(* IEC 61131-3 sources: advent-of-code/day10, 6 files *)

(* ---- demo.st ---- *)
VAR_GLOBAL CONSTANT
	str_len : DINT := 24; //Max length
	input_size : DINT := 9;
END_VAR

VAR_GLOBAL
	input : ARRAY[0..input_size-1] OF STRING[str_len];
END_VAR

FUNCTION set_input : __VOID
VAR_TEMP
	c : DINT;
END_VAR
	input[c] := '[({(<(())[]>[[{[]{<()<>>'; c := c + 1;
	input[c] := '[(()[<>])]({[<{<<[]>>('; c := c + 1;
	input[c] := '{([(<{}[<>[]}>{[]{[(<()>'; c := c + 1;
	input[c] := '(((({<>}<{<{<>}{[]{[]{}'; c := c + 1;
	input[c] := '[[<[([]))<([[{}[[()]]]'; c := c + 1;
	input[c] := '[{[{({}]{}}([{[{{{}}([]'; c := c + 1;
	input[c] := '{<[[]]>}<{[{[{[]{()[[[]'; c := c + 1;
	input[c] := '[<(<(<(<{}))><([]([]()'; c := c + 1;
	input[c] := '<{([([[(<>()){}]>(<<{{'; c := c + 1;
	input[c] := '<{([{{}}[<[[[<>{}]]]>[]]'; c := c + 1;
END_FUNCTION

(* ---- input.st ---- *)
VAR_GLOBAL CONSTANT
	str_len : DINT := 150; //Max length
	input_size : DINT := 110;
END_VAR

VAR_GLOBAL
	input : ARRAY[0..input_size-1] OF STRING[str_len];
END_VAR

FUNCTION set_input : __VOID
VAR_TEMP
	c : DINT;
END_VAR
input[c] := '<([<({{[<{{((<()>({}{})}<({}<>)>)}}>[<{(([()<>]<<>{}>))}<{({<>[]}<<>>)[([]<>)<{}{}>]}>>]]}}[<[{{[{{[<><>]'; c:= c+1;
input[c] := '[<{{{[((({<<<[()[]]{()()}><{<><>}(<>{})>><<{<><>}{{}[]}>{(()())[[]{}]}>>{[[(<>[]){<>{}}][(()())(()[])]]'; c:= c+1;
input[c] := '(((<{<[[<[{(((<><>)[{}{}]){{{}<>}[()<>]})(([<>()][<>{}]){{[]()}})}[({([][])<{}<>>}{[[]<>]{()'; c:= c+1;
input[c] := '[(<{<[<<<<[[{<[]()><<>()>}[{{}<>}<()>]]<<[[]{}]>{({}())}>]((((<>())<(){}>)<{[]{}}<(){}>>)[{[[]<>]<['; c:= c+1;
input[c] := '[[{(<{<<[{(<({<>{}}<()[]>){<<>[]>{<>}}><[[()[]]]{{()<>}{()<>}}])[{[(<>())]<<[]{}>(<>[])>}<[{'; c:= c+1;
input[c] := '(<<<[[<{({<<([{}{}](<><>)){{<><>}(())}>{<{(){}}{[][]}>[{[][]}([]())]}><([{{}[]}[[]{}]](<[]{}><{}<>>))((<(){'; c:= c+1;
input[c] := '<<<{((<<{[([<[[]{}]([][])>{[<>()][[][]]}]<<[()[]][[]{}]>[<<><>>(<><>)]>)<({{{}<>}{{}}}{{<><'; c:= c+1;
input[c] := '{[(<[{{{<[{({([]{}){{}{}}}[({}<>)])[([()[]]<[]{}>)<[{}{}]{{}()}>]}(<{{{}<>}(()[])}>{{<()<>><[]<>>}'; c:= c+1;
input[c] := '[<<{({[{((({<<<><>>(()())>{{[][]}<{}()>}}[[((){})[{}()]]<[()<>]>]){{(<{}<>>[()<>]){{[][]}(()<>'; c:= c+1;
input[c] := '({[([([<(<<[{<<><>>({}())}[[(){}][[][]]]]>><<(({<><>}{[][]})<{()()}[[]<>]>)[{((){}){{}[]}}(<<>()>{{}()})]><<'; c:= c+1;
input[c] := '[[[{[<({{<[[[<{}{}>(()())]{(<>[])([][])}]({{(){}}})]<[<{{}[]}{()}>[{<><>}]][<((){})([][])>]'; c:= c+1;
input[c] := '[(<{<{(<<<<{{[[][]]<()[]>}){{<<>{}>}}>({[(()())(<>[])]}(<{()()}[<>]>{[[]]<<>()>}))>(<[{({}{})}][{[{}()]'; c:= c+1;
input[c] := '<(<<[([[((<<{<[]{}>{{}<>}}(({}())[[]{}])>(<{<>()}[()()]>>>))]{<{{<(<()<>>{{}()})([{}<>](<><>))>'; c:= c+1;
input[c] := '[{[<[([[<[((([()[]]<{}{}>))<{[{}()][(){}]}([{}<>]<()<>>)>)]>[{((([{}()]{()()>)<(<><>)(()[])>)[(([]()'; c:= c+1;
input[c] := '{[{[{<<([({<<[{}()]<()<>>>{[[][]]({}())}>}[[<{{}<>}{<>}>]])(<<{[()[]]}(((){})({}{}))>[({{}()})]>)]('; c:= c+1;
input[c] := '({{{<<<<(([([[<><>]<<>[]>]{<()<>><()[]>})<([<>{}])>])(<<{{()}<()[]>}<([]<>)>>{{[{}()][[]<>]}[{<>}{()()'; c:= c+1;
input[c] := '[{(([{<{{(<{<<[]()>{{}<>}>}[<({}[])<{}<>>><{<>()}>]>)}<{{{{<<>{}>{()()}}}[[{()()}(()<>)><<{}<>>>]}[[(<(){}>('; c:= c+1;
input[c] := '[[{<[<(<[[<<({{}()}{{}})(({}{})[[]{}])>[([<>{}]({}<>))])]{<[<[[][]]<()<>>>]{([()()]{<><>})<{[]{}}[[]()]>}><'; c:= c+1;
input[c] := '([<<{({[({[({<{}[]>{{}<>}}){<[<>[]]>[(()())]}]{{{{{}[]>{()<>}}}<[{{}<>}<[]()>]([<>]<<><>>)>}})'; c:= c+1;
input[c] := '(([<[[{{(<[{{(()<>)}<<{}()>{<>{}}>}<[<[]()>[()()]]([<>()]{()})>)[(<[<><>]{{}<>}>{{{}()}{[]()}})<'; c:= c+1;
input[c] := '[([[[([[[<[{{<()()>{[][]}}(<[][]>)}[{<{}()>{<>[]}}]]>({[[{<><>}<[][]>]([()]{()[]})]}{([<<><>>[{}('; c:= c+1;
input[c] := '(<({<[[[[(((({[]{}}<{}<>>)[<(){}>[()<>]])){<(<<>{}>)<<()<>><()[]>>>{[[()()]<[][]>][{{}()}<<>{'; c:= c+1;
input[c] := '{{{{[[<{<{(<(([]())[{}[]])<(()<>){{}{}}}>){{{<{}[]><{}<>>}{(()[])[<><>]}}<{{()()}<<>[]>}>}}><(<[(<{'; c:= c+1;
input[c] := '<<[(<<<([{<{(({}())[{}[]])(<(){}>(<><>))}>([[(<>[])(<>[])]<({}{})<{}>>](((<>())<{}[]>)[[<>'; c:= c+1;
input[c] := '<{{((([[<{[(({<>{}}({}())))[([[]()][{}{}])]]}(([<([][])<<>()>>]<{{<>[]}(()())}[({}())[()()]]>)'; c:= c+1;
input[c] := '(({[{[[[[(<<[[(){}][(){}]]<{()<>}<[][])>>{({[][]}{<>{}}){<[][]>}}><{(([]{}){{}<>}){[()<>][('; c:= c+1;
input[c] := '{<[[<<([<{<<{[<>{}}{<><>}}(({}()))>[[{[]()}](<<>>{<><>})]><<([<>{}]{[][]})[<{}[]>{<><>}]>>}{[{(<<>()><{}<>'; c:= c+1;
input[c] := '({{{((({<<({<[<>()](()[])]}){((<{}()>{[]<>}){<[]{}>[[][]]})<[[[]{}](())](<{}<>>[{}])>}>[{{[(<>[])]}[<({}{'; c:= c+1;
input[c] := '{<(<[{({[[[{[[{}<>][(){}]]{{(){}}}}<<[[]()]{<>}><[{}[]]>>]{<<((){})[{}]>({<><>}{()[]})><<[{}()]{'; c:= c+1;
input[c] := '[[[(({<((<({<<{}>>}<[([]{})[[]]]>)<<{[()[]](<><>)}><<{[]{}}[[]]>{{()[]}{[]()}}>>><[((<(){}'; c:= c+1;
input[c] := '{{<{{{<<{<{<((<>[])<()[]>)<(<>{}){[][]}>><(({}<>){[][]}){[()<>]{<>{}}}>}>[((<<(){})({}())><([]'; c:= c+1;
input[c] := '[[[{({<[{[[<<(()<>)({}())>({<><>}[<><>])>]]<(<{<()<>>([]())}{[[]<>]{<>()}}>{<([][])((){})>([{}][()<>])})>}]<('; c:= c+1;
input[c] := '<<{[{[[<([[<<[{}<>]>[({}())<()[]>]>[{<(){}><{}<>>}[<<>>({}{})]]]<<{<()[]><()()>}({{}()}[{}<>])>>]<<([([]('; c:= c+1;
input[c] := '{<<<(<{{[{{{<<{}[]>{()()}>{[<>[]]({}())}}}<[<([]())>{<()()>(()())}][<(()())<{}<>>>((<><>)[[][]]]]>'; c:= c+1;
input[c] := '[[[({<(([[(<({()<>}<[]<>>)>[({[]}{<><>})<<(){}>{<><>}>])]]<(<[<<()()]<{}()>>(<{}()>([][]))]<<{<><>}>>>){'; c:= c+1;
input[c] := '<<[[<({<({[<{(()[])}{{[]()}<[]{}>}>]<[(<[]{}><<>{}>)<[()[]]([]{})>]>})>((<([<[<><>]([]{}}><{<>()}<()[]>>]{'; c:= c+1;
input[c] := '({[[[{{([[((<<{}<>}[{}<>]>)(({{}<>}<()()>)[[[]<>]<()<>>]))<(<{[][]}>)<{{[]<>}<[]<>>}[(<><>){(){}}]>>][<'; c:= c+1;
input[c] := '{<[[[[[<[[{{{{()}[[][]]}[<(){}>[[][]]]}(<[{}{}]>)}(<<<()()>{<>}>>)]<([[[()<>]((){})]([[]()]<{}{}>)]([{{}('; c:= c+1;
input[c] := '[<(({(((<[(<<[[]{}][<><>]>[{(){}}[[]]]><{{()[]}<<>()>}{{()}{(){}}}>)(<[([]())]<{{}{}}(())>>)]([([{()[]}[['; c:= c+1;
input[c] := '(({[([{{((({{<<>[]>}}<([{}[]][[]()])[{{}[]}<<>{}>]>)<({([])<[]{}>}){(((){})[<>[]]){<<>[]>[{}()'; c:= c+1;
input[c] := '<{<{(<<({([([([]())(<>[])][{()<>}{<>{}}])](({<()()>{()<>}}{{[]}[[][]]})[[[{}{}][()[]]]])]}(({[[{<>()}[{}()]'; c:= c+1;
input[c] := '[[{[{{[({<{<(<{}<>>)[[{}{}>[<><>]]>[((())([]<>)){([]())<<><>>}]}>{{{<{<>[]}({}{})>{([]{}){[][]}}}[{{<>'; c:= c+1;
input[c] := '[[{[<([{([<<<(<><>){[]{}}>{{[][]}([]<>)}>><{<<<>()>{<><>}>[<[][]>([]())]}({[{}[]]{<>()}}({()()}(()<>)))>])}])'; c:= c+1;
input[c] := '{{<((([<[({{(([]){[][]})[(()<>)<()()>]}{{{()[]}}([()[]][{}{}])}})<{({[()[]]<[]{}>}[<()()><()[]>])'; c:= c+1;
input[c] := '([<<<([{{<({{[{}<>][<>()]}{([]<>){(){}}}}){({<{}()>}[(()){<><>}])}><{<(<()[]>({}{}))(({}{})'; c:= c+1;
input[c] := '{{[([<[{<<{<{[{}[]][(){}]}[[[]()]{()[]}]>}><[(([<>{}]){{<>()}{()<>}}){[{<>{}}[[]<>]]{<[]<>>}}][[[{[]<'; c:= c+1;
input[c] := '{<<<<{(((<{([{{}{}}][[[]()]<<>()>])<([()<>]([]))[[<><>][{}()]]>}{<{{(){}}<()<>>}<{<>{}}{<>()}>>(<{'; c:= c+1;
input[c] := '<[({<{{{<((<<({})([]<>)>((<>[]){[]()}}>)(<[<(){}>({}[])]>[<({}<>){[][]}>[{()<>}<<><>>]]))>[({[([<>{}][{}()])<'; c:= c+1;
input[c] := '(({[[{<{[[((<[<>()]><{()<>}[[]<>]>)([{[]()}[[]()]](({}{}){<>()})>){<{(()())(<>[])}[<()[]>[()()]'; c:= c+1;
input[c] := '[(([{{<{<[{{{[{}{}]<(){}>}[<[]{}>({}())]}({[()[]]{[]()}}[<{}[]>(<>)])}[{{<[]{}>(()<>)}<[[]()]<<>[]>)}<<<<>()'; c:= c+1;
input[c] := '<(<<{<([([(<[{{}<>}<()()>][{()[]}(<><>)]>{{<[]<>><{}[]>>{{{}}{[]<>}}})({[<[]{}>[[][]]]}{{<'; c:= c+1;
input[c] := '((<<<([[<<{([<<>{}>{<>()}])<<{[]{}}[()[]]>>}[<{([]())[<>{}]}>{((()[]){{}<>))[<()<>>([]<>)]}]>{(({[[]]'; c:= c+1;
input[c] := '{<<((({({[<[[[<><>][<>{}]]{({}<>)<()[]>}][<<[]{}}<[]()>>[[[]<>]]]>([[[{}{}]]<<<><>><<>{}>>'; c:= c+1;
input[c] := '[{<([{{<{(<{{{(){}}{{}[]}}(<<>()>[()[]])}{{{{}}(()())}{[()<>]}}>[{[{[][]}{{}<>)]}((((){}){[]{}})(({})<<>{}'; c:= c+1;
input[c] := '[{[(<[{<{{[<{{()()}{()[]}}<<()()><{}[]>>>][<({()()}[()[]]){([][])[<>{}]}>(((()()))((<>{})<{}{'; c:= c+1;
input[c] := '(<(<([<<<{[<({<>}{()()})><((<>))<<{}[]><<><>>>>]{<{[[][]]}{{[]{}}{[]<>}>>[[[[]()]({})]]}}><<<<'; c:= c+1;
input[c] := '<([<(<<<(({{<[<><>]<[]<>>>(<[]()>[{}<>])}[<(()()){{}<>}>]}))<<[{{[<>[]]<()[]>}{(()<>){()()'; c:= c+1;
input[c] := '<[(<{{[[[<(([[<>()]([][])])){{{[()()]{{}[]}}[([]{}){(){}}]}{[<[]>{[]()}][[<>]({}())]}}>]]<(<[{<{<>()}{()['; c:= c+1;
input[c] := '<{{{[(<{<[<{{<()>(<>{})}[({}()){()()}]]([{<>{}}[()()]](<[]<>><<>{}>))>[<{<[]()>(<>)}<{[]{}}[('; c:= c+1;
input[c] := '<{(<[<[<{<({<[<><>}[[]()]>}([<(){}><<><>>][<()()><<><>>]))([[([]())<{}>]<[()()]{<>{}}>]{(({}'; c:= c+1;
input[c] := '<(<({(<[<[(((<<>{}>{{}()})){{[[]()](())}{{<><>}<<><>>}})([<<()()><[]())>[[<>()]<<>[]>]][<{()()}'; c:= c+1;
input[c] := '((<[{{(<[([<([()()](<>{}))(<{}()>[{}{}])>({<{}{}>(<>[])})])]>)}<({((([(<[]{}>({}[]))]{((<><>)(()()))}))(({{<{'; c:= c+1;
input[c] := '{({[<<[(<<((<<{}[]>[()<>]>{<<>[]>{[]()}}){[<<><>>[()[]]]<<{}()>[()<>]>})[{[{{}<>}{()}]}<(<()[]><{}{}>)[['; c:= c+1;
input[c] := '{{[<((<((<{[([[][]]<{}<>>)((()[]))]}>{[{(({}())[()[]]){{[][]}([][])}}](<<[<><>]{<>}><<{}<>><[][]>>>'; c:= c+1;
input[c] := '[[[<(<{{([{(<(<>{})(()<>)><(<>[])[{}()]>)([[[]()][[]<>]])}[[{<[]()>(<><>)}[(()){<>()}]]({{[]()}})]])[['; c:= c+1;
input[c] := '<({([{(<{{[<<[(){}][[]()>>[[{}{}](()[])]>]{{[[{}<>]{{}<>}]{({}<>)[{}{}]}}[({()()}[{}<>]){((){})}]}}{{[[{{'; c:= c+1;
input[c] := '[[[[{<[<(([<[<[]{}><<>{}>]<<[]<>>(()[])>>([(<>)<{}()>])])<{{({[]{}}{[]()})}<[[<><>]{[]<>}]{<<>()><<>()>}>'; c:= c+1;
input[c] := '<<<[([[(({(<[<{}>[{}()]]{{()}(()[]}}>(<<<>()>(<>[])>))<<[{<>()}{<>[]}][{[]{}}<{}[]>]>>}){<<<(<<>'; c:= c+1;
input[c] := '{{<[{{({{(([[([]{})<{}()>]]))){(<{{<<>[]>(<>[])}<<()><[]<>>>}>([([<>()]<{}[]>)(({}{}))]<<([]())[<>'; c:= c+1;
input[c] := '([<[({[{{[[[({<>{}}<(){}>)({<>[]}{()<>})](([(){}]{[]()}))]<[<(<>[])({}<>)>][[[[]{}]<()>]<<<>[]>{[]<>}>]>]'; c:= c+1;
input[c] := '{[{[[{<(<<({{([]<>)([]{})}<<{}<>><<>[]>>}(({()()}[{}()]){(<><>)[<>[]]]))<<[([])(<>[])]{([]())('; c:= c+1;
input[c] := '({<<{{[<<[{{<[(){}][[]]><{[]()}<[]{}>>}[<<<>()>{{}()}>[<{}<>>[<><>]]]}](<<[(<>{})[()]}{<<>><[]'; c:= c+1;
input[c] := '<<<([{[([{{[{[[]<>][<>[]]}]}{<([[][]]){[<>[]]<{}()>}><(<[]<>>(<>{}))[<[][]>{<>}]>}}{<{{[<>{}]{()'; c:= c+1;
input[c] := '<((<([([<{<[([{}<>](<>()))<([]<>)([]<>)>][<{()<>}{[]<>}>]>}<{[(<[]()>(<><>))[<(){}>[[][]]]](<([]())<<>[]>>['; c:= c+1;
input[c] := '{[<[<<{{(<{[{((){})<{}[]>}[([][])]]}{[({()<>}){[{}<>](<>{}))]}>)}<[[(<(<()<>>){(()())([]{})}>({[{}[]]'; c:= c+1;
input[c] := '<([[<({{[<({[({}{}){{}()}]<((){})[<><>]>})([[{[][]}<()<>>]<[()<>][{}{}]>])>]}}){{[(({(({[]()}{()()}'; c:= c+1;
input[c] := '<({([<[{(<[{(({}[]))}[[{[]<>}{{}[]}](({}[]))]]<[[(()[])[()()]]{[{}()>}]>>{<<{[[]<>](()())}[<{}[]>(<>'; c:= c+1;
input[c] := '(([[<(<<[{<(<[{}{}]{()<>}>)((<(){}>([]))({<>{}}[<>[]]))>(<<{()[]}{(){}}>[[<>()]]>[<{()[]}<()[]>>{({}<>){[]<'; c:= c+1;
input[c] := '{<[<<{(<{{<[{[{}()][<><>]}][{({}{})(<>[]))]>{<[[<><>]]<<<>()>({}[])>>({<[]<>>([]<>)}{[(){}]([]{})})'; c:= c+1;
input[c] := '{{<((([<{(([{[<>{}]{{}<>}}])<<<{<>[]}{(){}}>{(()[])[()[]]}>{{<<>()>}([(){}]{{}<>})}>)}{(([{{{}[]}(<>())'; c:= c+1;
input[c] := '{[(<{{{<[[{{[[()[]](<>{})]((()<>)({}[]))}}]][{([[{{}[]}<[]<>>]][{(<>{})}[(<>()){<><>}]])}>>[(['; c:= c+1;
input[c] := '<<<{([((<<{(({{}{}}({}{})))}{(<(<><>)[[]<>]>{[{}[]](<>)})<{{<>()}{{}<>}}<<<>[]><<>()>>>}>>))]){'; c:= c+1;
input[c] := '<{(<[[(({<[{{<<><>><{}<>>}<<<>{}>{()()}>}]>}))[((([([{[]{}}]([{}()][<><>]))(((<>())(<>]))]['; c:= c+1;
input[c] := '([<<[({(({{((<[]{}>{()[]}})({[<><>][<>()]}(<<><>>[[]()]))}{{{(()<>)({}{})}(<{}()><[]()>)}{{{<><>}'; c:= c+1;
input[c] := '[<<<{{<<{<{<<[()()](<><>)>>([({}){{}[]}]{<[]()>{{}()}})}<[{([]())<{}<>>}([{}()]<{}[]>)]<(<[]'; c:= c+1;
input[c] := '{{<[({({<{({((()<>)){[[]()]<(){}>>}<[[{}]{<><>}]<(()<>)<()()>>>)}(({((<><>)[{}[]]){[[]()][()[]]}})<({'; c:= c+1;
input[c] := '<[{<({<({(({{<(){}>[[]{}]}<<[][]><{}{}>>})[(([{}()][<>()]))[(<<>{}>([][]}){[[]{}]}]])[<[{(()<>)[{}<>]}]>]'; c:= c+1;
input[c] := '([(([{<(<{[<{([][]){[][]}}(<<>><[]{}>)>({[<>()]{{}<>}}(<<>[]>{<>{}}))][({{[]()}{[]}}(([]{})(()<>))'; c:= c+1;
input[c] := '<{<<<({[[(<<{(()<>)[[]{}]}<<()()>>>><[({()[]}[[][]]){<[][]>(<><>)}][(({}{})<()[]>){{{}()}<[]{}>}]>)[<((([]{}'; c:= c+1;
input[c] := '<([[([<<<{<<<<<><>>({}())>{{[]()}[{}[]]>>[<[<>()]({}{})>]>(({<{}{}>{<>{}}}{<{}[]>{{}()}}){[<[]()>{()<>}'; c:= c+1;
input[c] := '[{{<{[{{{<{{<([][])[()<>]>{{[]{}}({}())}}((<<>[]>([][])))}><{<<<{}<>><<>()>>{(()<>){[]{}}}>}{([{[][]}{<>{}}])'; c:= c+1;
input[c] := '[({<((({(<{[{<[][]}(<>[])}<<{}<>>{{}<>}>]({{<>()}[{}{}]})}(<{{{}()}<<>[]>}[([]{})<[][]>]>[{(<>'; c:= c+1;
input[c] := '<([[[<{{<<<[(((){})(()()))([<><>]{()})]<<[<>]([])>(([]<>))>>{{[<()>]<(()[])([][])>}[({{}}<{}{'; c:= c+1;
input[c] := '{<<((<[{<{<[{[[][]]{<><>}}{<(){}>{<><>}}]<((<>{})<<>[]>)>>((((<>[]){[]()})({<>()}))([[{}[]]{<>[]}]<'; c:= c+1;
input[c] := '(<{(<[[([[([<({}{})[()<>]>])][<{<({}())><{()()}>}>{[{[{}<>]([])}](([()()]))}]])]]>)}>[[({{'; c:= c+1;
input[c] := '(<[[[{<{[<([{({}{}){{}()}}[(<>{})<()()>]][{{{}()}}<{<>[]}[()<>]>]){{((<><>){()<>])<<<>()>[{}['; c:= c+1;
input[c] := '<{<<[((<<<{([{{}<>}({})]{((){})[[]<>]})<[[()<>]([]())](<[]<>>({}<>))>}{(<{()[]}>{<[]<>>})<'; c:= c+1;
input[c] := '{[([<[<[({{[<[<>()][{}[]}>((<>())<[]<>>)]{(<{}<>>(()()))([()()])}}}<(<(<<>{}>{<>{}})><({[]{}}['; c:= c+1;
input[c] := '{{[[[<<<<[[{({[]<>}<()()>)<<(){}>{<><>}>}{[([]<>)[<>[]]]}]{<[{()()}(<><>)]{{<>{}}<[]{}>}>((<{}()>{(){}}))}>>>'; c:= c+1;
input[c] := '({[<[[<{<([<<<()<>}<{}{}>>(<<>[]>(<>()))><{[<>()]({}<>)}<{[]{}}>>])>}{{{<{({[]{}}<<>>)<<[]<>'; c:= c+1;
input[c] := '([((((<(<[({((<>())<()<>>)}([<{}()>{<>()}]{{{}()}{[]<>)}))([<(<>{})><[(){}][<>()]>](([()]<[]{}>)(<{}{}>{()'; c:= c+1;
input[c] := '{[(<{({(<([(<[{}()][{}()]>)[[[{}()](()())]<{[][]}<[]<>>>]][({[()()]{{}{}}}((<><>)(<>())))<<{()()}{[]{}}}[{[]'; c:= c+1;
input[c] := '<([[{<<{<<{(([()<>]{<>[]})<<[][]>({}[])>)({<{}{}>([]<>)})}{<{{[][]}{[]{}}}[((){})((){})]><([[][]]){{()()}}>}'; c:= c+1;
input[c] := '(([<[[[(({{[[[[][]](<>())]{<<>><<>()>}]<<(()<>)>[<<>{}>{<><>}]>}[<(<<><>><{}{}>)[<()<>><[]()>]>[{<()[]>[<'; c:= c+1;
input[c] := '{[{{{[(<<[<[{[()()]<{}<>>}[([]<>)({}<>)]][<{()()}[<>[]]>]>]>>)]{([({[{({<>}(<>{}))[({}())[[][]]]}<{{()[]'; c:= c+1;
input[c] := '(<(<{<{<[[(({[<>[]]<{}[]>}[([]{})(()[])]))({([[]])([()()]{()[]})}<[<<><>><[]<>>]>)]]<([{{{{}<>}(<>)}}<({'; c:= c+1;
input[c] := '[<[{[<<[<<[<{<<>[]}<()>}{(()[])[{}[]]}><[<(){}>{{}[]}]>]>(((<{{}<>}{()[]}><<<>{}>{()[]}>)[[('; c:= c+1;
input[c] := '[<{(<[<{{([{{<<>{}><[]()>}({(){}}[[]{}])}{[<[][]>[<><>]][<<><>>[{}{}]]}](<<{(){}}({}<>)>(<()[]>[()[]])>'; c:= c+1;
input[c] := '<[{<({((([(<([[]<>]<()[]>)<(<>())>>(<{[][]>(<>{})>[{(){}}]))])))}<<{({<<<([]{})([]())>[{()()}<()<>>]'; c:= c+1;
input[c] := '<[(<{((({<<{{[{}<>]}[[<>{}]({}[])]}{(<{}[]}{<>})<{[]()}[()[]]>}>>}))(<<[<<(<<>{}><<>{}>)<<'; c:= c+1;
END_FUNCTION

(* ---- includes.st ---- *)
@EXTERNAL
FUNCTION printf : DINT
VAR_INPUT
str : STRING[1024];
params : ...;
END_VAR
END_FUNCTION

(* ---- sol.st ---- *)
FUNCTION main : DINT
	VAR_TEMP
		score  : DINT := 0;
		i : DINT := 0;
		completions : ARRAY[0..input_size-1] OF LINT;
		cmp_score : DINT := 0;
	END_VAR

	set_input();
	FOR i := 0 TO input_size-1 DO
		completions[i] := parse(&input[i]);
	END_FOR

	FOR i := 0 TO input_size-1 DO
		printf('%ld$n',completions[i]);
	END_FOR

END_FUNCTION

FUNCTION parse : LINT
VAR_INPUT
	str : REF_TO STRING[str_len];
END_VAR
VAR_TEMP
	current_str : Iterator;
	current_char : CHAR;
	letters : Stack;
END_VAR
		parse := 0;
		/* completion_score := 0; */
		current_str.set(str);
		WHILE current_str.has_next() DO
			//For each charachter in the string
			current_char := current_str.next();
			//If the charachter is an open char, add it to the stack
			IF is_open(current_char) THEN
				letters.push(current_char);
			ELSIF is_close(current_char) THEN //If it is a closing char: peek the top stack element
				IF get_pair(current_char) = letters.peek() THEN
					//If they match, pop
					letters.pop();
				ELSE
					//Otherwise break and score
					/* parse := score(current_char); */
					RETURN;
				END_IF
			END_IF
		END_WHILE
		//Anything remaining is a completion
		WHILE NOT letters.is_empty() DO
			parse := parse * 5 + score_cmp(get_pair(letters.pop()));
		END_WHILE

END_FUNCTION

FUNCTION get_pair : CHAR
VAR_INPUT
	c : CHAR;
END_VAR
	CASE c OF
		')': get_pair := '(';
		'(': get_pair := ')';
		']': get_pair := '[';
		'[': get_pair := ']';
		'{': get_pair := '}';
		'}': get_pair := '{';
		'>': get_pair := '<';
		'<': get_pair := '>';
	END_CASE
END_FUNCTION

FUNCTION is_open : BOOL
VAR_INPUT
	c : CHAR;
END_VAR
	CASE c OF
		'(','[','{','<' : is_open := TRUE;
	ELSE
		is_open := FALSE;
	END_CASE

END_FUNCTION

FUNCTION is_close : BOOL
VAR_INPUT
	c : CHAR;
END_VAR
	CASE c OF
		')',']','}','>' : is_close := TRUE;
	ELSE
		is_close := FALSE;
	END_CASE
END_FUNCTION

FUNCTION score : DINT
VAR_INPUT
	c : CHAR;
END_VAR
	score := 0;
	CASE c OF
		')': score := 3;
		']': score := 57;
		'}': score := 1197;
		'>': score := 25137;
	END_CASE
END_FUNCTION

FUNCTION score_cmp : LINT
VAR_INPUT
	c : CHAR;
END_VAR
	CASE c OF
		')': score_cmp := 1;
		']': score_cmp := 2;
		'}': score_cmp := 3;
		'>': score_cmp := 4;
	END_CASE
END_FUNCTION

(* ---- stack.st ---- *)
CLASS Stack
VAR
	arr : ARRAY[0..str_len] OF CHAR;
	counter : DINT := 0;
END_VAR

METHOD push : __VOID
	VAR_INPUT
		p : CHAR;
	END_VAR
	arr[counter] := p;
	counter := counter + 1;
END_METHOD

METHOD pop : CHAR
	counter := counter - 1;
	IF counter < 0 THEN
		counter := 0;
	END_IF
	pop := arr[counter];
END_METHOD

METHOD peek : CHAR
	peek := arr[counter - 1];
END_METHOD

METHOD is_empty : BOOL
	is_empty := counter = 0;
END_METHOD

END_CLASS

(* ---- str.st ---- *)
(* A string iterator class *)
CLASS Iterator
	VAR
		str : REF_TO STRING[str_len];
		counter : DINT := 0;
	END_VAR

	METHOD set : __VOID
		VAR_INPUT
			val : REF_TO STRING;
		END_VAR
		str := val;
		counter := 0;
	END_METHOD

	METHOD next : CHAR
	VAR_TEMP
		ptr : REF_TO CHAR;
		ptr_val : LWORD;
	END_VAR
		ptr := str;
		ptr_val := ptr;
		ptr_val := ptr_val + counter;
		ptr := ptr_val;
		next := ptr^;
		/* printf('Next at %d : %c$n',counter, next); */

		counter := counter + 1;
	END_METHOD

	METHOD has_next : BOOL
	VAR_TEMP
		ptr : REF_TO CHAR;
		ptr_val : LWORD;
	END_VAR
		ptr := str;
		ptr_val := ptr;
		ptr_val := ptr_val + counter;
		ptr := ptr_val;

		has_next := ptr^ <> 0 AND counter < str_len+1;
	END_METHOD

END_CLASS
